// Get information from a mover using this structure
TYPE StationDict :
STRUCT
    StationNum : INT;
    StationPos : LREAL;
END_STRUCT
END_TYPE

(* stored: Version 1.1.0.1, ProductVersion 3.1.4024.12
   DUT StationDict: Id {7f3cd863-6356-409d-a480-336d9d9a09b4} *)
